(* Funzione che calcola l'ingombro della pinza nelle varie dimensioni a seconda del ciclo che la massima sta eseguendo *)
FUNCTION TFCalcoliIngombroPinza_ConAsseK : BOOL
VAR_INPUT

	Mission : POINTER TO TFMachinePalletizer_Mission;
	WorkAreaManager : POINTER TO TFWorkAreaManager;
	//
	AngoloRotazioneDestinazionePinza : LREAL; //Ango di rotazione del quale si vogliono calcolare le quote degli ingombri a destinazione  
	ModuleAX_J : POINTER TO TFModulePalletizer_AxJ_Lastre;//Modulo Asse rotazione
	//
	AngoloRotazioneDestinazionePiano : LREAL; //Angolo di rotazione del piano della pinza DESTINAZIONE => 90° = pinza parallela all'asse X
	ModuleAX_K : POINTER TO TFModulePalletizer_AxJ_Lastre;//Modulo Asse rotazione PIANO

	IngombroX_Pos : POINTER TO LREAL;//Ingombro della pinza nella Metà POSITIVA della pinza lungo X
	IngombroY_Pos : POINTER TO LREAL;//Ingombro della pinza nella Metà POSITIVA della pinza lungo Y
	
	IngombroX_Neg : POINTER TO LREAL;//Ingombro della pinza nella Metà NEGATIVA della pinza lungo X
	IngombroY_Neg : POINTER TO LREAL;//Ingombro della pinza nella Metà NEGATIVA della pinza lungo Y
	
	IngombroY_Tot : POINTER TO LREAL;//Ingombro totale In direzione Y
	
	IngombroZ_Pos : POINTER TO LREAL;//Ingombro della pinza lungo Z Positivo (sopra al fulcro)
	IngombroZ_Neg : POINTER TO LREAL;//Ingombro della pinza lungo Z Negativo (sotto al fulcro)
	
	IngombroDestinazioneX_Pos : POINTER TO LREAL;//Ingombro della pinza nella Metà POSITIVA della pinza lungo X
	IngombroDestinazioneY_Pos : POINTER TO LREAL;//Ingombro della pinza nella Metà POSITIVA della pinza lungo Y
	
	IngombroDestinazioneX_Neg : POINTER TO LREAL;//Ingombro della pinza nella Metà NEGATIVA della pinza lungo X
	IngombroDestinazioneY_Neg : POINTER TO LREAL;//Ingombro della pinza nella Metà NEGATIVA della pinza lungo Y
	
	IngombroDestinazioneZ_Pos : POINTER TO LREAL;//Ingombro della pinza lungo Z Positivo (sopra al fulcro)
	IngombroDestinazioneZ_Neg : POINTER TO LREAL;//Ingombro della pinza lungo Z Negativo (sotto al fulcro)
	
	IngombroMaxX_Pos : POINTER TO LREAL;//Ingombro MASSIMO della pinza nella Metà POSITIVA della pinza lungo X
	IngombroMaxY_Pos : POINTER TO LREAL;//Ingombro MASSIMO della pinza nella Metà POSITIVA della pinza lungo Y
	
	IngombroMaxX_Neg : POINTER TO LREAL;//Ingombro MASSIMO della pinza nella Metà NEGATIVA della pinza lungo X
	IngombroMaxY_Neg : POINTER TO LREAL;//Ingombro MASSIMO della pinza nella Metà NEGATIVA della pinza lungo Y
	
	IngombroMaxZ_Pos : POINTER TO LREAL;//Ingombro MASSIMO della pinza lungo Z Positivo (sopra al fulcro)
	IngombroMaxZ_Neg : POINTER TO LREAL;//Ingombro MASSIMO della pinza lungo Z Negativo (sotto al fulcro)

	IngombroY_Pos_0 : POINTER TO LREAL;//Ingombro della pinza nella Metà POSITIVA della pinza lungo Y
	IngombroY_Neg_180 : POINTER TO LREAL;//Ingombro della pinza nella Metà NEGATIVA della pinza lungo Y
	IngombroY_Neg_0 : POINTER TO LREAL;//Ingombro della pinza nella Metà POSITIVA della pinza lungo Y
	IngombroY_Pos_180 : POINTER TO LREAL;//Ingombro della pinza nella Metà NEGATIVA della pinza lungo Y
		
	ScostamentoVerticalePuntoCentrale : POINTER TO LREAL; //Valore che rappresenta quanto il punto centrale si è spostato rispetto allo zero orizzontale (lungo Z crescente)
END_VAR

VAR
	LunghezzaMAX 	: LREAL;//LunghezzaMAX Totale pinza
	LarghezzaMAX 	: LREAL;//Larghezza Totale pinza
	SpessoreMAX  	: LREAL;//Spessore Totale pinza	
	DimTraveVerticale : LREAL; //Dimensione Trave/Ingombro Centrale

	Diagonale			: LREAL;
	MezzaDiagonale   	: LREAL;
	Lx_MezzoAttuale : LREAL;
	Ly_MezzoAttuale : LREAL;
	Lx_MezzoDest : LREAL;
	Ly_MezzoDest : LREAL;
	Beta : LREAL;
	AngoloPerCalcoloRotPianoAttuale 	 : LREAL;
	AngoloPerCalcoloRotPianoDestinazione : LREAL;


END_VAR

(* Calcolo delle dimensioni della pinza in base al tipo di ciclo in corso *)
CASE WorkAreaManager^.State OF
	WAMANAGER_NOP,
	
	WAMANAGER_CICLO_RIPOSO_INIT:
		SpessoreMAX 	:= Dimensioni_Pinza.Spessore;
		LunghezzaMAX 	:= Dimensioni_Pinza.Lunghezza;
		LarghezzaMAX    := Dimensioni_Pinza.Larghezza;
		
	WAMANAGER_CICLO_RIPOSO_RUN:
		
		SpessoreMAX 	:= Dimensioni_Pinza.Spessore;
		LunghezzaMAX 	:= Dimensioni_Pinza.Lunghezza;
		LarghezzaMAX    := Dimensioni_Pinza.Larghezza;
															
	WAMANAGER_CICLO_PRELIEVO_FALDA_RUN:
	
		SpessoreMAX 	:= Dimensioni_Pinza.Spessore;
		LunghezzaMAX 	:= Dimensioni_Pinza.Lunghezza;
		LarghezzaMAX    := Dimensioni_Pinza.Larghezza;

	WAMANAGER_CICLO_DEPOSITO_FALDA_RUN:
		
		SpessoreMAX 	:= Dimensioni_Pinza.Spessore;
		LunghezzaMAX 	:= MAX(Dimensioni_Pinza.Lunghezza,Mission^.XDim);
		LarghezzaMAX    := MAX(Dimensioni_Pinza.Larghezza,Mission^.YDim);
										

	WAMANAGER_CICLO_PRELIEVO_LASTRA_WA_RUN:
		SpessoreMAX 	:= Dimensioni_Pinza.Spessore;
		LunghezzaMAX 	:= Dimensioni_Pinza.Lunghezza;
		LarghezzaMAX    := Dimensioni_Pinza.Larghezza;
					
	WAMANAGER_CICLO_DEPOSITO_LASTRA_SU_PAREGGIATORE_RUN:
		SpessoreMAX 	:= Dimensioni_Pinza.Spessore;
		LunghezzaMAX 	:= MAX(Dimensioni_Pinza.Lunghezza,Mission^.XDim);
		LarghezzaMAX    := MAX(Dimensioni_Pinza.Larghezza,Mission^.YDim);
					
	WAMANAGER_CICLO_PRELIEVO_LASTRA_DA_PAREGGIATORE_RUN:
	
		SpessoreMAX 	:= Dimensioni_Pinza.Spessore;
		LunghezzaMAX 	:= Dimensioni_Pinza.Lunghezza;
		LarghezzaMAX    := Dimensioni_Pinza.Larghezza;
								
	WAMANAGER_CICLO_DEPOSITO_LASTRA_WA_RUN:
	
		SpessoreMAX 	:= Dimensioni_Pinza.Spessore;
		LunghezzaMAX 	:= MAX(Dimensioni_Pinza.Lunghezza,Mission^.XDim);
		LarghezzaMAX    := MAX(Dimensioni_Pinza.Larghezza,Mission^.YDim);

	WAMANAGER_CICLO_LASTRA_PP_INIT:
		SpessoreMAX 	:= Dimensioni_Pinza.Spessore;
		LunghezzaMAX 	:= Dimensioni_Pinza.Lunghezza;
		LarghezzaMAX    := Dimensioni_Pinza.Larghezza;
						
	WAMANAGER_CICLO_PRELIEVO_LASTRA_PP_RUN:
	
		SpessoreMAX 	:= Dimensioni_Pinza.Spessore;
		LunghezzaMAX 	:= Dimensioni_Pinza.Lunghezza;
		LarghezzaMAX    := Dimensioni_Pinza.Larghezza;
						
	WAMANAGER_CICLO_DEPOSITO_LASTRA_PP_RUN:
	
		SpessoreMAX 	:= Dimensioni_Pinza.Spessore;
		LunghezzaMAX 	:= MAX(Dimensioni_Pinza.Lunghezza,Mission^.XDim);
		LarghezzaMAX    := MAX(Dimensioni_Pinza.Larghezza,Mission^.YDim);

	(* Ciclo lastra per depalettizzare da postazioni senza formature, con autoapprndimenti*)
	WAMANAGER_CICLO_PRELIEVO_LASTRA_DEPAL_RUN :
	
		SpessoreMAX 	:= Dimensioni_Pinza.Spessore;
		LunghezzaMAX 	:= Dimensioni_Pinza.Lunghezza;
		LarghezzaMAX    := Dimensioni_Pinza.Larghezza;
																				
	(* Ciclo lastra deposito su rulliera *)
	WAMANAGER_CICLO_DEPOSITO_LASTRA_DEPAL_RUN :
	
		SpessoreMAX 	:= Dimensioni_Pinza.Spessore;
		LunghezzaMAX 	:= MAX(Dimensioni_Pinza.Lunghezza,Mission^.XDim);
		LarghezzaMAX    := MAX(Dimensioni_Pinza.Larghezza,Mission^.YDim);
													
	(* Ciclo deposito FALDA su magazzino dedicato *)
	WAMANAGER_CICLO_DEPOSITO_FALDA_DEPAL_RUN :
	
		SpessoreMAX 	:= Dimensioni_Pinza.Spessore;
		LunghezzaMAX 	:= MAX(Dimensioni_Pinza.Lunghezza,Mission^.XDim);
		LarghezzaMAX    := MAX(Dimensioni_Pinza.Larghezza,Mission^.YDim);

	(* Ciclo PRELIEVO DA PANCONE *)
	WAMANAGER_CICLO_PRELIEVO_LASTRA_DA_PANCONE_RUN:
	
		SpessoreMAX 	:= Dimensioni_Pinza.Spessore;
		LunghezzaMAX 	:= Dimensioni_Pinza.Lunghezza;
		LarghezzaMAX    := Dimensioni_Pinza.Larghezza;

	(* Ciclo DEPOSITO SU PANCONE *)
	WAMANAGER_CICLO_DEPOSITO_LASTRA_SU_PANCONE_RUN:
	
		SpessoreMAX 	:= Dimensioni_Pinza.Spessore;
		LunghezzaMAX 	:= MAX(Dimensioni_Pinza.Lunghezza,Mission^.XDim);
		LarghezzaMAX    := MAX(Dimensioni_Pinza.Larghezza,Mission^.YDim);

	(* Ciclo PRELIEVO DA CANTILEVER *)
	WAMANAGER_CICLO_PRELIEVO_LASTRA_DA_CANTILEVER_RUN:
	
		SpessoreMAX 	:= Dimensioni_Pinza.Spessore;
		LunghezzaMAX 	:= Dimensioni_Pinza.Lunghezza;
		LarghezzaMAX    := Dimensioni_Pinza.Larghezza;

	(* Ciclo DEPOSITO SU CANTILEVER *)
	WAMANAGER_CICLO_DEPOSITO_LASTRA_SU_CANTILEVER_RUN:
	
		SpessoreMAX 	:= Dimensioni_Pinza.Spessore;
		LunghezzaMAX 	:= MAX(Dimensioni_Pinza.Lunghezza,Mission^.XDim);
		LarghezzaMAX    := MAX(Dimensioni_Pinza.Larghezza,Mission^.YDim);

	(* Ciclo DEPOSITO SU CANTILEVER *)
	WAMANAGER_CICLO_POSIZIONAMENTO_SEMPLICE_RUN:
	
		SpessoreMAX 	:= Dimensioni_Pinza.Spessore;
		LunghezzaMAX 	:= Dimensioni_Pinza.Lunghezza;
		LarghezzaMAX    := Dimensioni_Pinza.Larghezza;
ELSE
	SpessoreMAX 	:= Dimensioni_Pinza.Spessore;
	LunghezzaMAX 	:= MAX(Dimensioni_Pinza.Lunghezza,Mission^.XDim);
	LarghezzaMAX    := MAX(Dimensioni_Pinza.Larghezza,Mission^.YDim);
END_CASE

DimTraveVerticale := Dimensioni_Pinza.DimTraveVerticale;


Diagonale		:= SQRT(LunghezzaMAX*LunghezzaMAX+LarghezzaMAX*LarghezzaMAX);//Diagonale lastra
MezzaDiagonale	:= Diagonale/2; //Metà diagonale lastra	
Beta 			:= ATAN((LarghezzaMAX/2)/(LunghezzaMAX/2));	//Angolo dato dalla diagonale
//
AngoloPerCalcoloRotPianoAttuale := Beta + deg_to_rad(ModuleAX_K^.Ax^.AxRef^.NcToPlc.ActPos);

(* Calcolo lungo X e lungo Y i valori di ingombro a seconda di come è ruotato il piano della pinza *)
Lx_MezzoAttuale		:= ABS(MezzaDiagonale * COS(AngoloPerCalcoloRotPianoAttuale-(PI/2))); //Metà Lato "LX" parallelo all'asse X con lastra in piano
Ly_MezzoAttuale		:= ABS(MezzaDiagonale * SIN(AngoloPerCalcoloRotPianoAttuale-(PI/2))); //Metà Lato "LY" parallelo all'asse Y con lastra in piano

(* Calcolo gli ingombri in base al'angolo di rotazione della pinza *)
//IngombroX_Pos^ 	:=  LunghezzaMAX/2;
//IngombroX_Neg^ 	:=  LunghezzaMAX/2;
IngombroX_Pos^ 	:=  Lx_MezzoAttuale;// LunghezzaMAX/2;
IngombroX_Neg^ 	:=  Lx_MezzoAttuale;// LunghezzaMAX/2;


IngombroY_Neg^ 	:= MAX((Ly_MezzoAttuale * COS(deg_to_rad(-90+ModuleAX_J^.Ax^.AxRef^.NcToPlc.ActPos)) +
					SpessoreMAX * SIN(deg_to_rad(-90+ModuleAX_J^.Ax^.AxRef^.NcToPlc.ActPos))),DimTraveVerticale/2);
					
IngombroY_Pos^ 	:= ABS(MIN((-Ly_MezzoAttuale * COS(deg_to_rad(-90+ModuleAX_J^.Ax^.AxRef^.NcToPlc.ActPos)) +
					SpessoreMAX * SIN(deg_to_rad(-90+ModuleAX_J^.Ax^.AxRef^.NcToPlc.ActPos))),DimTraveVerticale/2));	

(* In base a come la pinza è ruotata inverto il positivo con il negativo in modo da avere sempre i valori corretti *)
IF AngoloRotazioneDestinazionePinza < 90 THEN	                         
	IngombroZ_Pos^	:= ABS(((Ly_MezzoAttuale) * SIN(deg_to_rad(-90+ModuleAX_J^.Ax^.AxRef^.NcToPlc.ActPos)))+
									(SpessoreMAX * COS(deg_to_rad(-90+ModuleAX_J^.Ax^.AxRef^.NcToPlc.ActPos)))-SpessoreMAX);

	IngombroZ_Neg^	:= ABS((-(Ly_MezzoAttuale) * SIN(deg_to_rad(-90+ModuleAX_J^.Ax^.AxRef^.NcToPlc.ActPos))) +
									(SpessoreMAX * COS(deg_to_rad(-90+ModuleAX_J^.Ax^.AxRef^.NcToPlc.ActPos)))-SpessoreMAX);

ELSIF  AngoloRotazioneDestinazionePinza > 90 THEN					
	IngombroZ_Pos^	:= ABS((-(Ly_MezzoAttuale) * SIN(deg_to_rad(-90+ModuleAX_J^.Ax^.AxRef^.NcToPlc.ActPos))) +
									(SpessoreMAX * COS(deg_to_rad(-90+ModuleAX_J^.Ax^.AxRef^.NcToPlc.ActPos)))-SpessoreMAX);	
	IngombroZ_Neg^	:= ABS(((Ly_MezzoAttuale) * SIN(deg_to_rad(-90+ModuleAX_J^.Ax^.AxRef^.NcToPlc.ActPos)))+
								(SpessoreMAX * COS(deg_to_rad(-90+ModuleAX_J^.Ax^.AxRef^.NcToPlc.ActPos)))-SpessoreMAX);
ELSE
	IngombroZ_Pos^	:= ABS(((Ly_MezzoAttuale) * SIN(deg_to_rad(-90+ModuleAX_J^.Ax^.AxRef^.NcToPlc.ActPos)))+
									(SpessoreMAX * COS(deg_to_rad(-90+ModuleAX_J^.Ax^.AxRef^.NcToPlc.ActPos)))-SpessoreMAX);

	IngombroZ_Neg^	:= ABS((-(Ly_MezzoAttuale) * SIN(deg_to_rad(-90+ModuleAX_J^.Ax^.AxRef^.NcToPlc.ActPos))) +
									(SpessoreMAX * COS(deg_to_rad(-90+ModuleAX_J^.Ax^.AxRef^.NcToPlc.ActPos)))-SpessoreMAX);
END_IF
IngombroY_Tot := IngombroY_Pos + IngombroY_Neg;//Ingombro TOTALE in direzione Y


(* Calcolo gli ingombri in base al'angolo di rotazione FINALE *)
AngoloPerCalcoloRotPianoDestinazione := Beta + deg_to_rad(AngoloRotazioneDestinazionePiano);

(* Calcolo lungo X e lungo Y i valori di ingombro a seconda di come è ruotato il piano della pinza *)
Lx_MezzoDest	:= ABS(MezzaDiagonale * COS(AngoloPerCalcoloRotPianoDestinazione-(PI/2))); //Metà Lato "LX" parallelo all'asse X con lastra in piano
Ly_MezzoDest	:= ABS(MezzaDiagonale * SIN(AngoloPerCalcoloRotPianoDestinazione-(PI/2))); //Metà Lato "LY" parallelo all'asse Y con lastra in piano

IngombroDestinazioneX_Pos^ 	:= Lx_MezzoDest;//  LunghezzaMAX/2;
IngombroDestinazioneX_Neg^ 	:= Ly_MezzoDest;// LunghezzaMAX/2;

IngombroDestinazioneY_Neg^ 	:= MAX((Ly_MezzoDest * COS(deg_to_rad(-90+AngoloRotazioneDestinazionePinza)) +
									SpessoreMAX * SIN(deg_to_rad(-90+AngoloRotazioneDestinazionePinza))),DimTraveVerticale/2);
					
IngombroDestinazioneY_Pos^ 	:= ABS(MIN((-Ly_MezzoDest * COS(deg_to_rad(-90+AngoloRotazioneDestinazionePinza)) +
									SpessoreMAX * SIN(deg_to_rad(-90+AngoloRotazioneDestinazionePinza))),DimTraveVerticale/2));
	
(* In base a come la pinza è ruotata inverto il positivo con il negativo in modo da avere sempre i valori corretti *)
IF AngoloRotazioneDestinazionePinza < 90 THEN	                         
	IngombroDestinazioneZ_Pos^	:= ABS(((Ly_MezzoDest) * SIN(deg_to_rad(-90+AngoloRotazioneDestinazionePinza)))+
									(SpessoreMAX * COS(deg_to_rad(-90+AngoloRotazioneDestinazionePinza)))-SpessoreMAX);

	IngombroDestinazioneZ_Neg^	:= ABS((-(Ly_MezzoDest) * SIN(deg_to_rad(-90+AngoloRotazioneDestinazionePinza))) +
									(SpessoreMAX * COS(deg_to_rad(-90+AngoloRotazioneDestinazionePinza)))-SpessoreMAX);

ELSIF  AngoloRotazioneDestinazionePinza > 90 THEN					
	IngombroDestinazioneZ_Pos^	:= ABS((-(Ly_MezzoDest) * SIN(deg_to_rad(-90+AngoloRotazioneDestinazionePinza))) +
									(SpessoreMAX * COS(deg_to_rad(-90+AngoloRotazioneDestinazionePinza)))-SpessoreMAX);	
	IngombroDestinazioneZ_Neg^	:= ABS(((Ly_MezzoDest) * SIN(deg_to_rad(-90+AngoloRotazioneDestinazionePinza)))+
								(SpessoreMAX * COS(deg_to_rad(-90+AngoloRotazioneDestinazionePinza)))-SpessoreMAX);
ELSE
	IngombroDestinazioneZ_Pos^	:= ABS(((Ly_MezzoDest) * SIN(deg_to_rad(-90+AngoloRotazioneDestinazionePinza)))+
									(SpessoreMAX * COS(deg_to_rad(-90+AngoloRotazioneDestinazionePinza)))-SpessoreMAX);

	IngombroDestinazioneZ_Neg^	:= ABS((-(Ly_MezzoDest) * SIN(deg_to_rad(-90+AngoloRotazioneDestinazionePinza))) +
									(SpessoreMAX * COS(deg_to_rad(-90+AngoloRotazioneDestinazionePinza)))-SpessoreMAX);
END_IF

(* Calcolo degli ingombri massimi nelle varie dimensioni *)
IngombroMaxX_Pos^ := MAX(IngombroX_Pos^,IngombroDestinazioneX_Pos^);//Ingombro MASSIMO della pinza nella Metà POSITIVA della pinza lungo X
IngombroMaxY_Pos^ := MAX(IngombroY_Pos^,IngombroDestinazioneY_Pos^);//Ingombro MASSIMO della pinza nella Metà POSITIVA della pinza lungo Y

IngombroMaxX_Neg^ := MAX(IngombroX_Neg^,IngombroDestinazioneX_Neg^);//Ingombro MASSIMO della pinza nella Metà NEGATIVA della pinza lungo X
IngombroMaxY_Neg^ := MAX(IngombroY_Neg^,IngombroDestinazioneY_Neg^);//Ingombro MASSIMO della pinza nella Metà NEGATIVA della pinza lungo Y

IngombroMaxZ_Pos^ := MAX(IngombroZ_Pos^,IngombroDestinazioneZ_Pos^);//Ingombro MASSIMO della pinza lungo Z Positivo (sopra al fulcro)
IngombroMaxZ_Neg^ := MAX(IngombroZ_Neg^,IngombroDestinazioneZ_Neg^);//Ingombro MASSIMO della pinza lungo Z Negativo (sotto al fulcro)


/////////////////////////////

IngombroY_Pos_0^ := ABS(MIN(SpessoreMAX * SIN(deg_to_rad(-90)),DimTraveVerticale/2));
IngombroY_Neg_180^ := ABS(MAX(SpessoreMAX * SIN(deg_to_rad(-90+180)),DimTraveVerticale/2));

IngombroY_Neg_0^ := ABS(MAX(SpessoreMAX * SIN(deg_to_rad(-90)),DimTraveVerticale/2));
IngombroY_Pos_180^ := ABS(MIN(SpessoreMAX * SIN(deg_to_rad(-90+180)),DimTraveVerticale/2));
								
ScostamentoVerticalePuntoCentrale^ := ABS(SpessoreMAX * COS(deg_to_rad(-90+AngoloRotazioneDestinazionePinza))-SpessoreMAX);
																
TFCalcoliIngombroPinza := TRUE;

END_FUNCTION

(* stored: Version 1.1.0.1, ProductVersion 3.1.4024.11
   POU TFCalcoliIngombroPinza_ConAsseK: Id {00bc9d52-bca1-4f9a-8acd-fe33e115ddda}, SpecialFunc None *)
